FUNCTION_BLOCK FB_CASE_FinaliseDataTests EXTENDS TcUnit.FB_TestSuite

//==============================================================
//MAIN TESTS
//==============================================================

test01_();

METHOD INTERNAL test01_
VAR
	fbCase		: FB_CASE_FinaliseData;	
END_VAR
TcUnit.TEST('test01_');

fbCase(
	bExecute:= , 
	stProductInstruction:= , 
	stPackCodesDuplicated:= , 
	stOuterBarcodeDuplicate:= , 
	stOuterDuplicatedPackCodesFound:= , 
	stCaseRejectReasons:= , 
	stCACData:= , 
	bDone=> , 
	bBusy=> , 
	bCACValid=> , 
	sRejectCode=> , 
	bIsDuplicateOuters=> , 
	bIsDuplicatePacks=> , 
	bReadyToValidate=> , 
	stUpdateCACData=> 
);

TEST_FINISHED();
END_METHOD

END_FUNCTION_BLOCK

(* stored: Version 1.1.0.1
   POU FB_CASE_FinaliseDataTests: Id {97469738-e6cc-4ef5-9bb6-76a47206d06d}, SpecialFunc None
   Method test01_: Id {994630ca-cb5c-49c7-9f2d-af6c76c304fa} *)
